# EPICS substitutions: iocBoot/iocArcusMotor/motor.substitutions
file "$(MOTOR)/db/basic_asyn_motor.db"
{
pattern
{P,           N,   M,      DTYP,        PORT, ADDR, DESC,       EGU, DIR,   VELO,  VBAS, ACCL, BDST, BVEL, BACC, MRES, PREC,   DHLM,   DLLM, INIT}
{MOT:, 1,    "m$(N)", "asynMotor",  "P0",   0,    "Screen $(N)", in,  Pos,   1,     0,    0.2,  0,    1,    0.2,  0.0001, 2,      3,      -3,   ""}
}
